{attribute 'linkalways'} 
{attribute 'no_explicit_call' := 'This FB is a CLASS and must be accessed using methods or properties'}
{attribute 'enable_dynamic_creation'}
FUNCTION_BLOCK Stack EXTENDS Disposable
VAR
	linkedList : LinkedList;
END_VAR

METHOD PUBLIC Clear
VAR_INPUT
END_VAR
linkedList.Clear();
END_METHOD

METHOD PUBLIC Contains : BOOL;
VAR_INPUT
	Item : ANY;
END_VAR
VAR
	found : I_LinkedListNode;
END_VAR
found := linkedList.Find(Item);
Contains := found <> 0;
END_METHOD

METHOD PUBLIC CopyTo : BOOL
VAR_INPUT
	Destination : ANY;
END_VAR
CopyTo := linkedList.CopyTo(Destination);
END_METHOD

METHOD PUBLIC CopyToLocation : BOOL
VAR_INPUT
	Destination : PVOID;
	DestinationSize : UDINT;
END_VAR
CopyToLocation := linkedList.CopyToLocation(Destination,DestinationSize);
END_METHOD

PROPERTY PUBLIC Count : ULINT
GET
Count := linkedList.Count;
END_GET
END_PROPERTY

METHOD PUBLIC GetEnumerator : I_ForwardEnumerator
GetEnumerator := linkedList.GetEnumerator();
END_METHOD

METHOD PROTECTED OnDispose : BOOL
VAR_INPUT
    CalledExplicitly : BOOL; // true if disposal was triggered from Dispose()
END_VAR
Clear();
END_METHOD

METHOD PUBLIC Push
VAR_INPUT
	Item : ANY;
END_VAR
linkedList.AddFirst(Item);
END_METHOD

METHOD PUBLIC TryPeek : BOOL;
VAR_INPUT
	Destination : ANY;
END_VAR
VAR
	first : I_LinkedListNode;
END_VAR
first := linkedList.First;

IF first = 0 THEN
	RETURN;
END_IF

TryPeek := first.Get(Destination);
END_METHOD

METHOD PUBLIC TryPop : BOOL;
VAR_INPUT
	Destination : ANY;
END_VAR
VAR
	first : I_LinkedListNode;
	popped : BOOL;
END_VAR
first := linkedList.First;

IF first = 0 THEN
	RETURN;
END_IF

popped := linkedList.First.Get(Destination);

IF NOT popped THEN
	RETURN;
END_IF

linkedList.RemoveFirst();
TryPop := TRUE;
END_METHOD

END_FUNCTION_BLOCK

(* stored: Version 1.1.0.1, ProductVersion 3.1.4024.12
   POU Stack: Id {4790b190-51f0-4629-938e-d46fbfba08da}, SpecialFunc None
   Folder Protected: Id {cfbdc69c-c35e-47df-9655-8180f0a6b883}
   Method Clear: Id {75e9b203-44b9-46cb-9b54-1e02ee5d7b99}
   Method Contains: Id {380b1f79-30ca-466a-8058-741c367b1b90}
   Method CopyTo: Id {af958370-a50e-4e86-9c4b-ff6a7cc7410a}
   Method CopyToLocation: Id {28903e4e-8156-4bd6-b962-c02c0a27e37c}
   Property Count: Id {a94a5378-7530-4234-b8d6-9da634e0e108}
   Get Get: Id {32f5b2ef-b4fc-43f9-8efb-27f1fb752ef0}
   Method GetEnumerator: Id {40757687-c6f0-426e-be33-fde6ea7dbab6}
   Method OnDispose: Id {c7d4f371-0cdc-4589-a504-8d46e1406072}
   Method Push: Id {1a16ddc8-f918-4565-8544-bf1a2ae21019}
   Method TryPeek: Id {e0200c18-235c-43fd-8c04-d6e1cbe0445e}
   Method TryPop: Id {5057eaf3-9ed3-4dc9-ada0-912b0844cda6} *)
